INTERFACE I_MqttMessageReceiver

METHOD OnMqttMessage : BOOL
VAR_INPUT
	rMqttMessage : REFERENCE TO FB_IotMqttMessage;
END_VAR
END_METHOD

END_INTERFACE

(* stored: Version 1.1.0.1, ProductVersion 3.1.4024.5
   Itf I_MqttMessageReceiver: Id {44a731eb-092a-4e6b-b9a6-a9847f702b69}
   Method OnMqttMessage: Id {993a4ddc-f32b-46f5-bda1-504ff5b3e3df} *)
